FUNCTION_BLOCK TimeChannelParametersFB
VAR_INPUT
END_VAR
VAR_OUTPUT
END_VAR
VAR
END_VAR

END_FUNCTION_BLOCK

(* stored: Version 1.1.0.1, ProductVersion 3.1.4024.6
   POU TimeChannelParametersFB: Id {da56f15f-511d-409e-bbc6-3822c1ef44b4}, SpecialFunc None *)
